// TwinCAT 3 PLC project Riverside
// ProgramVersion: 3.1.4023.0
// libraries:
//   EfficientIO Communicator, * (EfficientIO)
//   EfficientIO Energy Basic, * (EfficientIO)
//   Lynus HTTP Functions, * (Lynus AG)
//   Lynus Standards, * (EfficientIO)
//   Tc2_Standard, * (Beckhoff Automation GmbH)
//   Tc2_System, * (Beckhoff Automation GmbH)
//   Tc3_Module, * (Beckhoff Automation GmbH)
// project tree:
//   FBs/ FB_SPOpt_Monitoring_extTime.TcPOU
//   POUs/ MAIN.TcPOU, prgCom.TcPOU, prgLynus.TcPOU
//   / Riverside_Fast.TcTTO, Riverside_Middle.TcTTO
// (motion and I/O tree: see PLC project untitled1)
// real-time tasks:
//   TASK PlcTask: cycle T#10ms, priority 10, ADS port 350
//   TASK Com: cycle T#20ms, priority 14, ADS port 352
//   TASK Lynus: cycle T#5ms, priority 6, ADS port 351
//   TASK Riverside_Fast: cycle T#5ms, priority 8, ADS port 353
//   TASK Riverside_Middle: cycle T#20ms, priority 12, ADS port 354

CONFIGURATION Riverside
    RESOURCE PLC ON TwinCAT3
        TASK Riverside_Fast(INTERVAL := T#5ms, PRIORITY := 8);
        TASK Riverside_Middle(INTERVAL := T#20ms, PRIORITY := 12);
        PROGRAM MAIN WITH Riverside_Fast : MAIN;
        PROGRAM prgLynus WITH Riverside_Fast : prgLynus;
        PROGRAM prgCom WITH Riverside_Middle : prgCom;
    END_RESOURCE
END_CONFIGURATION

// ---- POUs/MAIN.TcPOU
PROGRAM MAIN
VAR
	fbVarInfo						: FB_VarInfo;	
	timStart						: TON;
	timResetConnection				: TON;
	byLPArr							: BYTE;
	iState							: INT;	
	uiErrorCounter					: UINT;
	fbMonitor						: FB_SPOpt_Monitoring_extTime;
	bSEnableOp						: BOOL;			//{#lynus.ag#()}
	rHeartbeat						: REAL;			//{#lynus.ag#()}
	rErrorWarning					: REAL;			//{#lynus.ag#()}
	rSPOptReady						: REAL;			//{#lynus.ag#()}
	rNewTargetValue					: REAL;			//{#lynus.ag#()} //Optimierter Sollwert Vorlauftemperatur
	byHB							: BYTE;			//Watchdog
	FPStart							: R_TRIG;
	FPDone							: R_TRIG;
	FPError							: R_TRIG;
	fbHttp							: FB_GetSet_Data_Auhofcenter;
		
	x: INT;

	// Riverside
	rRiverside_AT					: REAL;			//{#lynus.ag#()}
	rRiverside_VL					: REAL;			//{#lynus.ag#()}
	rRiverside_RL					: REAL;			//{#lynus.ag#()}
	rRiverside_EGPalmers			: REAL;			//{#lynus.ag#()}
	rRiverside_EGNanuNana			: REAL;			//{#lynus.ag#()}
	rRiverside_EGKindOptik			: REAL;			//{#lynus.ag#()}
	rRiverside_EGBijouBrigitte		: REAL;			//{#lynus.ag#()}
	rRiverside_OGGlaskubus			: REAL;			//{#lynus.ag#()}
	rRiverside_OGMediaMarkt			: REAL;			//{#lynus.ag#()}
	rRiverside_OGDepot				: REAL;			//{#lynus.ag#()}
	rRiverside_OGRauwolf			: REAL;			//{#lynus.ag#()}
	rRiverside_OGYuzu				: REAL;			//{#lynus.ag#()}

	Timer_Wait: Ton;
	
	bDissableExtHBRIV : BOOL;			//{#lynus.ag#()}
END_VAR
VAR PERSISTENT
	bEnableWrite					: BOOL:=TRUE;		
	bEnableOp						: BOOL;			//{#lynus.ag#()}
END_VAR

//Search the Variabels for Lynus
fbVarInfo(
	bReadInfo:= , 
	eTMCFile:= eSelectTMCFile.eDontUseTMCFile, 
	eSavePositionTMCFile:= eSavePositionOnPLC.ePostionC, 
	udiCounterFoundVariables=> , 
	bError=> , 
	bBusy=> , 
	byProgress=> , 
	udiErrorCodeOut=> , 
	eErrorVarInfo_Out=> , 
	sVarWithError=> );

//Monitor
fbMonitor(
	bEnable:= bEnableOp, 
	bDissableHB:= TRUE, 
	tChangeHBIn:= T#1H, 
	tChangeHBOut:= T#30S, 
	rHeartbeat:= rHeartbeat, 
	rErrorWarning:= rErrorWarning, 
	rSPOptReady:= rSPOptReady,
	bReadyOut=> , 
	bDissableExtHB=> bDissableExtHBRIV, 
	bSEnable=> bSEnableOp, 
	rHeartbeatOut=> );
	
//Read/Write Function to the Auhofcenter System	
timStart(IN:= TRUE, PT:= T#5S, Q=> , ET=> );

FPStart(CLK:= timStart.Q, Q=> );

IF FPStart.Q THEN
	iState := 1;	
END_IF

CASE iState OF

	0://Stop
		fbHttp.bStart := FALSE;

	1://Read Values
		fbHttp.bStart := TRUE;	
			fbHttp.bReadRequest := TRUE;
				fbHttp.bWriteRequest := FALSE;
		
		// Riverside
		//DV900 Aussentemperatur °C
		x:=1;
		fbHttp.arrListOfVariables[x].bIsString := FALSE;
		fbHttp.arrListOfVariables[x].sVariableName := 'DV900';	
		fbHttp.arrListOfVariables[x].sVariableValue := '';
		//DV911 Riverside Vorlauftemperatur °C
		x:=2;
		fbHttp.arrListOfVariables[x].bIsString := FALSE;
		fbHttp.arrListOfVariables[x].sVariableName := 'DV911';	
		fbHttp.arrListOfVariables[x].sVariableValue := '';
		//DV912 Riverside Rücklauftemperatur °C
		x:=3;
		fbHttp.arrListOfVariables[x].bIsString := FALSE;
		fbHttp.arrListOfVariables[x].sVariableName := 'DV912';	
		fbHttp.arrListOfVariables[x].sVariableValue := '';
		//DV921 Riverside Raumtemperatur Mall EG, vor Palmers °C
		x:=4;
		fbHttp.arrListOfVariables[x].bIsString := FALSE;
		fbHttp.arrListOfVariables[x].sVariableName := 'DV921';	
		fbHttp.arrListOfVariables[x].sVariableValue := '';
		//DV922 Riverside Raumtemperatur Mall EG, vor Nanu-Nana °C
		x:=5;
		fbHttp.arrListOfVariables[x].bIsString := FALSE;
		fbHttp.arrListOfVariables[x].sVariableName := 'DV922';	
		fbHttp.arrListOfVariables[x].sVariableValue := '';
		//DV923 Riverside Raumtemperatur Mall EG, vor Kind Optik °C
		x:=6;
		fbHttp.arrListOfVariables[x].bIsString := FALSE;
		fbHttp.arrListOfVariables[x].sVariableName := 'DV923';
		fbHttp.arrListOfVariables[x].sVariableValue := '';
		//DV924 Riverside Raumtemperatur Mall EG, vor Bijou Brigitte °C
		x:=7;
		fbHttp.arrListOfVariables[x].bIsString := FALSE;
		fbHttp.arrListOfVariables[x].sVariableName := 'DV924';	
		fbHttp.arrListOfVariables[x].sVariableValue := '';
		//DV925 Riverside Raumtemperatur Mall 1. OG, Glaskubus °C
		x:=8;
		fbHttp.arrListOfVariables[x].bIsString := FALSE;
		fbHttp.arrListOfVariables[x].sVariableName := 'DV925';	
		fbHttp.arrListOfVariables[x].sVariableValue := '';
		//DV926 Riverside Raumtemperatur Mall 1. OG, vor Media Markt °C
		x:=9;
		fbHttp.arrListOfVariables[x].bIsString := FALSE;
		fbHttp.arrListOfVariables[x].sVariableName := 'DV926';	
		fbHttp.arrListOfVariables[x].sVariableValue := '';
		//DV927 Riverside Raumtemperatur Mall 1. OG, vor Depot °C
		x:=10;
		fbHttp.arrListOfVariables[x].bIsString := FALSE;
		fbHttp.arrListOfVariables[x].sVariableName := 'DV927';	
		fbHttp.arrListOfVariables[x].sVariableValue := '';
		//DV928 Riverside Raumtemperatur Mall 1. OG, vor Rauwolf °C
		x:=11;
		fbHttp.arrListOfVariables[x].bIsString := FALSE;
		fbHttp.arrListOfVariables[x].sVariableName := 'DV928';	
		fbHttp.arrListOfVariables[x].sVariableValue := '';
		//DV929 Riverside Raumtemperatur Mall 1. OG, vor Yuzu °C
		x:=12;
		fbHttp.arrListOfVariables[x].bIsString := FALSE;
		fbHttp.arrListOfVariables[x].sVariableName := 'DV929';	
		fbHttp.arrListOfVariables[x].sVariableValue := '';
(*		//
		x:=;
		fbHttp.arrListOfVariables[x].bIsString := FALSE;
		fbHttp.arrListOfVariables[x].sVariableName := '';	
		fbHttp.arrListOfVariables[x].sVariableValue := '';
*)				
		IF FPDone.Q THEN 
			iState := 3; 
				//Auf Lynus Variablen mappen
				(*-----------Riverside----------------*)
				rRiverside_AT	:= STRING_TO_REAL(fbHttp.arrListOfVariabelsOut[1].sVariableValue);
				rRiverside_VL	:= STRING_TO_REAL(fbHttp.arrListOfVariabelsOut[2].sVariableValue);
				rRiverside_RL	:= STRING_TO_REAL(fbHttp.arrListOfVariabelsOut[3].sVariableValue);
				rRiverside_EGPalmers	:= STRING_TO_REAL(fbHttp.arrListOfVariabelsOut[4].sVariableValue);
				rRiverside_EGNanuNana	:= STRING_TO_REAL(fbHttp.arrListOfVariabelsOut[5].sVariableValue);
				rRiverside_EGKindOptik	:= STRING_TO_REAL(fbHttp.arrListOfVariabelsOut[6].sVariableValue);
				rRiverside_EGBijouBrigitte	:= STRING_TO_REAL(fbHttp.arrListOfVariabelsOut[7].sVariableValue);
				rRiverside_OGGlaskubus	:= STRING_TO_REAL(fbHttp.arrListOfVariabelsOut[8].sVariableValue);
				rRiverside_OGMediaMarkt	:= STRING_TO_REAL(fbHttp.arrListOfVariabelsOut[9].sVariableValue);
				rRiverside_OGDepot	:= STRING_TO_REAL(fbHttp.arrListOfVariabelsOut[10].sVariableValue);
				rRiverside_OGRauwolf	:= STRING_TO_REAL(fbHttp.arrListOfVariabelsOut[11].sVariableValue);
				rRiverside_OGYuzu	:= STRING_TO_REAL(fbHttp.arrListOfVariabelsOut[12].sVariableValue);
		END_IF
			IF FPError.Q THEN iState := 300; END_IF


	3://wait state
		Timer_Wait.IN := TRUE;
		IF bEnableWrite AND Timer_Wait.Q THEN
			Timer_Wait.IN := FALSE;
			iState := 4; 
		ELSIF  Timer_Wait.Q THEN
			Timer_Wait.IN := FALSE;
			iState := 1; 
		END_IF
		
	4://Write Values
	
		// clear array
		FOR byLPArr := 1 TO 100 BY 1 DO
			fbHttp.arrListOfVariables[byLPArr].bIsString := FALSE;
			fbHttp.arrListOfVariables[byLPArr].sVariableName := '';	
			fbHttp.arrListOfVariables[byLPArr].sVariableValue := '';	
		END_FOR
		
		IF fbMonitor.bDissableExtHB THEN byHB := 0; END_IF

	
		fbHttp.bStart := TRUE;	
		fbHttp.bReadRequest := FALSE;
		fbHttp.bWriteRequest := TRUE;
					
		
		//Watchdog
		fbHttp.arrListOfVariables[1].bIsString := FALSE;
		fbHttp.arrListOfVariables[1].sVariableName := 'DV931';
		fbHttp.arrListOfVariables[1].sVariableValue := REAL_TO_STRING(BYTE_TO_REAL(byHB));		
	
		// Heinzung aus/Ein
		fbHttp.arrListOfVariables[2].bIsString := FALSE;
		fbHttp.arrListOfVariables[2].sVariableName := 'DV932';
		fbHttp.arrListOfVariables[2].sVariableValue := '1';	

		//Neuer Sollwert für den Vorlauf für die Regelung
		fbHttp.arrListOfVariables[3].bIsString := FALSE;
		fbHttp.arrListOfVariables[3].sVariableName := 'DV933';
		fbHttp.arrListOfVariables[3].sVariableValue := REAL_TO_STRING(rNewTargetValue);	
		
				
		IF FPDone.Q THEN 
			iState := 5; 
				IF NOT fbMonitor.bDissableExtHB THEN byHB := byHB + 1; END_IF
		END_IF
			IF FPError.Q THEN 
				iState := 300; 
				IF NOT fbMonitor.bDissableExtHB THEN byHB := byHB + 1; END_IF
			END_IF
			
		IF byHB > 1 THEN byHB := 0; END_IF
	5://wait state
		Timer_Wait.IN := TRUE;
		IF Timer_Wait.Q THEN
			Timer_Wait.IN := FALSE;
			iState := 1; 
		END_IF		
	300://Error
		uiErrorCounter := uiErrorCounter + 1;
			iState := 1; 
			
END_CASE

fbHttp(
	bStart:= , 
	bWriteRequest:= , 
	bReadRequest:= , 
	tDelayRequest:= T#10S, 
	sHostname:= '172.24.17.110', 
	arrListOfVariables:= , 
	bValidResult=> , 
	bBusy=> , 
	bError=> , 
	bDone=> , 
	arrListOfVariabelsOut=> , 
	hrErrorCode=> );
	
FPDone(CLK:= fbHttp.bDone, Q=> );
	FPError(CLK:= fbHttp.bError, Q=> );

Timer_Wait(PT:=T#5S);

END_PROGRAM

// ---- FBs/FB_SPOpt_Monitoring_extTime.TcPOU
{attribute 'hide_all_locals'}
FUNCTION_BLOCK FB_SPOpt_Monitoring_extTime
VAR_INPUT PERSISTENT
	bEnable							: BOOL;									//{#lynus.ag#()} //Enable or dissable thsi function
	bDissableHB						: BOOL;									//If this is True, then the Output HB is also dissabled when we have a Error or the Ready Flag from the Backend Service is not OK. If its False the HB is only dissalbed when the Function is not Enables or the HB from the Backend Service is missing
	tChangeHBIn						: TIME := T#70S;						//Delay bettwen the changes from the HB at the Input HB Variable
	tChangeHBOut					: TIME := T#30S;						//Delay bettwen the changes from the HB at the Output HB Variable
END_VAR
VAR_INPUT
	rHeartbeat						: REAL;									//{#lynus.ag#()} //Heartbeat from the Service. NOT OVERRIDE
	rErrorWarning					: REAL;									//{#lynus.ag#()} //Error or Warning from the Service. NOT OVERRIDE
	rSPOptReady						: REAL;									//{#lynus.ag#()} //Setpoint Optimization Service Ready. NOT OVERRIDE
END_VAR
VAR_OUTPUT
	bError							: BOOL;									//Error from this Fuction
	bReadyOut						: BOOL;									//Show if the Service is Read or not
	bDissableExtHB					: BOOL;									//If someone use a external HB with this Flag he can see if the HB, ready or Error Flag from the Backend is set
	bSEnable						: BOOL;									//{#lynus.ag#()} //Enable State of hte function
	rHeartbeatOut					: REAL;									//Heartbeat for the external Service
	diNrOfSPOpt_OUT					: DINT;									//Active Number from Setpoint Optimizer for using on other functions
END_VAR
VAR
	rHBInput_CP						: REAL;									//Variable to compare input HB Variable to set or reset the timer
	fbNumberDevice					: FB_NumberOfDevice;					//Function block to calcualte the number of the Device
	timDissableFunctions			: TON;									//Timer to dissable the Function after Lynus_Standards.Constants_General.tTimeDissableLynusFunctions Days without connection to the Lynus Cloud
	timResetConnectionOnGVL			: TON;									//Timer to try reset the connection Flag on the GVL. (When somebody delete the Connection Function and make only a onlinechange)
	timHBInput						: TON;									//Timer to check the Input HB
	timHBOutput						: TON;									//Timer to set the Output HB
	timReady						: TON;									//Timer to dissable the Ready Flag
	timErrorWarning					: TON;									//Timmer do detect a Error or a Warning
END_VAR

//Creator : Kai Ebensperger
//Company : Lynus AG
//Date : 03.12.2021
//Version : 1.0.0.0

//This is a Function for using with the Setpoin Optimizer on our Backen System.
//So we have the possibility to send the Ready Flag and the HB to the external system we are communicating with in the right intervals.  
//Error evaluation also takes place in this function. Thus, in the event of an error or other event, the Ready flag, the HB or even both can be deactivated and the external system can switch back to classic control. 


(*-------------------------------------------------------------------------------Limits----------------------------------------------------------------------------------------------*)

rHeartbeat := LIMIT(0,rHeartbeat,1);
	rErrorWarning := LIMIT(0,rErrorWarning,2);
		rSPOptReady := LIMIT(0,rSPOptReady,1);
			tChangeHBIn := LIMIT(T#1S,tChangeHBIn,T#1H); // increased this max-Limit due to issues at Cloud-SPO
				tChangeHBOut := LIMIT(T#1S,tChangeHBOut,T#600S);	
	
(*-------------------------------------------------------------Calcualte the number of SP Opttimizer---------------------------------------------------------------*)

fbNumberDevice(
	diActualNumberOfDevices:= Lynus_Standards.GVL_Energy.stNumberOfDevices.diNumberOfSetPointOpt, 
	diMaxNumberOfDevices:= Constants_Energy.diMaxNumberOfSetPointOpt, 
	udiCounterOnlineChange:= TwinCAT_SystemInfoVarList._AppInfo.OnlineChangeCnt, 
	bNumberIsCalculatet=> , 
	bFPNumberIsCalculatet=> , 
	bOnlineChange=> , 
	diNumberForThisDevice=> diNrOfSPOpt_OUT, 
	diNumberOfTotalDevices=> );

//Write new Numer on GVL
IF fbNumberDevice.bFPNumberIsCalculatet THEN
	Lynus_Standards.GVL_Energy.stNumberOfDevices.diNumberOfSetPointOpt := fbNumberDevice.diNumberOfTotalDevices;	
END_IF 

//Delete old Number on GVL
IF fbNumberDevice.bOnlineChange THEN 
	Lynus_Standards.GVL_Energy.stNumberOfDevices.diNumberOfSetPointOpt := diNrOfSPOpt_OUT;
END_IF			
			
(*-------------------------------------------------------------Service from Backend is ready and check the connection to backen for dissabel/enable EMS Function---------------------------------------------------------------*)

//Try to reset the variable for connection on the GVL. When all is normal then the Lynus Mqtt connection function set this variable to true in the next cycle
//When we have no connection to the backend or no HB from the Service then after Lynus_Standards.Constants_General.tTimeDissableLynusFunctions days the EMS is dissabled with all of his functionalities
timResetConnectionOnGVL(IN:= NOT timResetConnectionOnGVL.Q, PT:= T#1H, Q=> , ET=> );
	IF timResetConnectionOnGVL.Q THEN Lynus_Standards.GVL_Communicator.bStateConnectionToEnableFunctions := FALSE; END_IF
		IF NOT Lynus_Standards.GVL_Communicator.bStateConnectionToEnableFunctions OR rHBInput_CP = rHeartbeat THEN timDissableFunctions.IN := TRUE; ELSE timDissableFunctions.IN := FALSE; END_IF  
			timDissableFunctions(IN:= , PT:= Lynus_Standards.Constants_General.tTimeDissableLynusFunctions, Q=> , ET=> );

(*------------------------------------------------------------------Error----------------------------------------------------------------------------*)	

IF Lynus_Standards.GVL_Energy.stNumberOfDevices.diNumberOfSetPointOpt > Constants_Energy.diMaxNumberOfSetPointOpt THEN bError := TRUE; ELSE bError := FALSE; END_IF 
			
(*-----------------------------------------------------------------------------------------------------Logic--------------------------------------------------------------------------------------------------------------*)

bSEnable := bEnable;

//Input HB
timHBInput(IN:= , PT:= tChangeHBIn, Q=> , ET=> );
	IF rHeartbeat <> rHBInput_CP THEN
		timHBInput.IN := FALSE; rHBInput_CP := rHeartbeat;
	ELSE
		timHBInput.IN := TRUE;
	END_IF

//Ready
IF rSPOptReady = 0 THEN timReady.IN := TRUE; ELSE timReady.IN := FALSE; END_IF
	timReady(IN:= , PT:= tChangeHBIn * 2, Q=> , ET=> ); 	
	
//Error and Warning
IF rErrorWarning <> 0 THEN timErrorWarning.IN := TRUE; ELSE timErrorWarning.IN := FALSE; END_IF
	timErrorWarning(IN:= , PT:= tChangeHBIn * 2, Q=> , ET=> );
	
//Set HB Output and Ready Flag
IF rSPOptReady <> 0 AND NOT timReady.Q AND bEnable AND NOT timDissableFunctions.Q AND NOT timErrorWarning.Q THEN bReadyOut := TRUE; END_IF
	IF timReady.Q OR timErrorWarning.Q THEN bReadyOut := FALSE; END_IF

IF (NOT timHBInput.Q AND bDissableHB AND bReadyOut AND NOT timErrorWarning.Q AND NOT timHBOutput.Q AND bEnable AND NOT timDissableFunctions.Q) OR
	(NOT timHBInput.Q AND NOT bDissableHB AND NOT timHBOutput.Q AND bEnable AND NOT timDissableFunctions.Q) THEN
		timHBOutput.IN := TRUE;
ELSE
		timHBOutput.IN := FALSE;
END_IF
	timHBOutput(IN:= , PT:= tChangeHBOut, Q=> , ET=> );
		IF timHBOutput.Q THEN rHeartbeatOut := rHeartbeatOut + 1; END_IF
 			IF rHeartbeatOut > 1 THEN rHeartbeatOut := 0; END_IF

//External HB Flag
IF timHBInput.Q OR (timReady.Q AND bDissableHB) OR (timErrorWarning.Q AND bDissableHB) THEN
	bDissableExtHB := TRUE;
ELSE
	bDissableExtHB := FALSE;
END_IF   
	
//Not Enabled
IF NOT bEnable OR timDissableFunctions.Q OR bError THEN
	bReadyOut := FALSE;
		bDissableExtHB := TRUE;
			rHeartbeatOut := 0;	
END_IF

END_FUNCTION_BLOCK

// ---- POUs/prgLynus.TcPOU
PROGRAM prgLynus
VAR
	fbRW1		: FB_ReadWrite_V2;
END_VAR

fbRW1(
	eUploadType:= eSelectDataUploadType.e_Change_Intervall5min , 
	bBusy=> , 
	bError=> , 
	udiErrorCodeOut=> , 
	eErrorReadWrite_Out=> );

END_PROGRAM

// ---- POUs/prgCom.TcPOU
PROGRAM prgCom
VAR
	fbCom			: FB_MqttCommunicator_V5;
END_VAR

fbCom(
	bConnect:= TRUE, 
	strAuthKey:=  'ENE87365342998' ,
	sUserName:= '55a5520b-7d81-4677-a7f3-53eed27dacea', 
	sUserPassword:= '16d1c65b-166e-486f-a478-f0c72de3f9ce', 
	eSavePositionCertificate:= eSavePositionOnPLC.ePostionC, 
	time_HeartBeat_sec := T#1S,
	bConnected=> , 
	bError=> , 
	hrErrorCode=> , 
	eConnectionState=> , 
	eErrorMessage_Out=> );

END_PROGRAM
